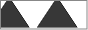
VISUALIZATION Valve  // 88x30
VAR_IN_OUT
	valve_toggleColor : BOOL;
	valve_tapVariable : BOOL;
END_VAR
    Polygon (37,27) (57,-3) (77,27) (66,27) (52,27), colour toggle: valve_toggleColor
        tap valve_tapVariable
    Polygon (-11,27) (9,-3) (29,27) (18,27) (4,27), colour toggle: valve_toggleColor
        tap valve_tapVariable
END_VISUALIZATION

(* stored: Version 1.1.0.1, ProductVersion 3.1.4024.9
   Visu Valve: Id {28baef22-0d1a-4521-9c50-57d98c0ec5ea} *)
